// TIA Portal project "Ejercicio4-Proceso-TIA" (V14)

(* hardware
DEVICE "S7-1200 station_1"  S7-1200 Station
   slot 0: "Rack_0"  S7-1200 Rack  Rack  V1.0
   slot 1: "PLC_1"  CPU 1214C AC/DC/Rly  6ES7 214-1BG40-0XB0  V4.2
   slot 2: "AI 4x13BIT_1"  SM 1231 AI4  6ES7 231-4HD30-0XB0  V1.0
DEVICE "HMI_1"  TP 277 6''
   slot 0: "TP 277 6''"  TP 277 6''  6AV6 643-0AA01-1AX0  11.0.2.0
   slot 1: "HMI_RT_1"  TP 277 6''  6AV6 643-0AA01-1AX0  11.0.2.0
   slot 5: "HMI_1.IE_CP_1"  PROFINET Interface  11.0.0.0
      slot 1: "Interfaz PROFINET_1"  PROFINET Interface
         slot 1: "Port_1"  Port
   slot 7: "HMI_1.MPI/DP_CP_1"  MPI/DP Interface  11.0.0.0
*)

// ===== PLC "PLC_1"  CPU 1214C AC/DC/Rly =====

VAR_GLOBAL   // PLC tag table "Tabla de variables estándar"
   "System_Byte" AT %MB1 : Byte;
   "FirstScan" AT %M1.0 : Bool;
   "DiagStatusUpdate" AT %M1.1 : Bool;
   "AlwaysTRUE" AT %M1.2 : Bool;
   "AlwaysFALSE" AT %M1.3 : Bool;
   "System_Byte(1)" AT %MB1 : Byte;
   "Clock_Byte" AT %MB100 : Byte;
   "Clock_10Hz" AT %M100.0 : Bool;
   "Clock_5Hz" AT %M100.1 : Bool;
   "Clock_2.5Hz" AT %M100.2 : Bool;
   "Clock_2Hz" AT %M100.3 : Bool;
   "Clock_1.25Hz" AT %M100.4 : Bool;
   "Clock_1Hz" AT %M100.5 : Bool;
   "Clock_0.625Hz" AT %M100.6 : Bool;
   "Clock_0.5Hz" AT %M100.7 : Bool;
   "Tag_2" AT %MD8 : Real;
   "LT1" AT %IW30 : Int;
   "TT1" AT %IW100 : Int;
   "TT2" AT %IW102 : Int;
   "TT3" AT %IW104 : Int;
   "LT2" AT %IW98 : Int;
   "SLT1" AT %MD30 : Real;
   "SLT2" AT %MD38 : Real;
   "STT1" AT %MD46 : Real;
   "STT2" AT %MD54 : Real;
   "LedLT1" AT %Q0.0 : Bool;
   "LedLT2" AT %Q0.1 : Bool;
   "LedTT1" AT %Q0.2 : Bool;
   "LedTT2" AT %Q0.3 : Bool;
   "CorteDeLazo" AT %M0.5 : Bool;
   "START" AT %M0.0 : Bool;
   "STOP" AT %M0.1 : Bool;
   "Salida" AT %QD30 : Real;
   "Entrada" AT %ID2 : Real;
   "EncenderTanque" AT %ID6 : Real;
   "Ldl" AT %Q0.4 : Bool;
   "START/STOP" AT %M0.3 : Bool;
END_VAR

DATA_BLOCK "Transmisor TT1"   // DB1
{ S7_Optimized_Access := 'TRUE' }
VERSION : 0.1
// stored: InstanceOfName Escalado
"Escalado"
BEGIN
END_DATA_BLOCK

DATA_BLOCK "Transmisor TT2"   // DB2
{ S7_Optimized_Access := 'TRUE' }
VERSION : 0.1
// stored: InstanceOfName Escalado
"Escalado"
BEGIN
END_DATA_BLOCK

DATA_BLOCK "Transmisor LT1"   // DB3
{ S7_Optimized_Access := 'TRUE' }
VERSION : 0.1
// stored: InstanceOfName Escalado
"Escalado"
BEGIN
END_DATA_BLOCK

DATA_BLOCK "Transmisor LT2"   // DB4
{ S7_Optimized_Access := 'TRUE' }
VERSION : 0.1
// stored: InstanceOfName Escalado
"Escalado"
BEGIN
END_DATA_BLOCK

FUNCTION_BLOCK "Escalado"   // FB1, LAD
TITLE = Bloque de Escalado en Tension
{ S7_Optimized_Access := 'TRUE' }
VERSION : 0.1
   VAR_INPUT
      Entrada_IV : Int;
      ISH : Int;
      ISL : Int;
      OSH : Real;
      OSL : Real;
   END_VAR
   VAR_OUTPUT
      Salida : Real;
   END_VAR
   VAR_TEMP
      Temp_D : DInt;
      Temp_R : Real;
   END_VAR
BEGIN

REGION Network 1
   // (OSH - OSL)*(IV-ISL)/(ISH-ISL)+OSL
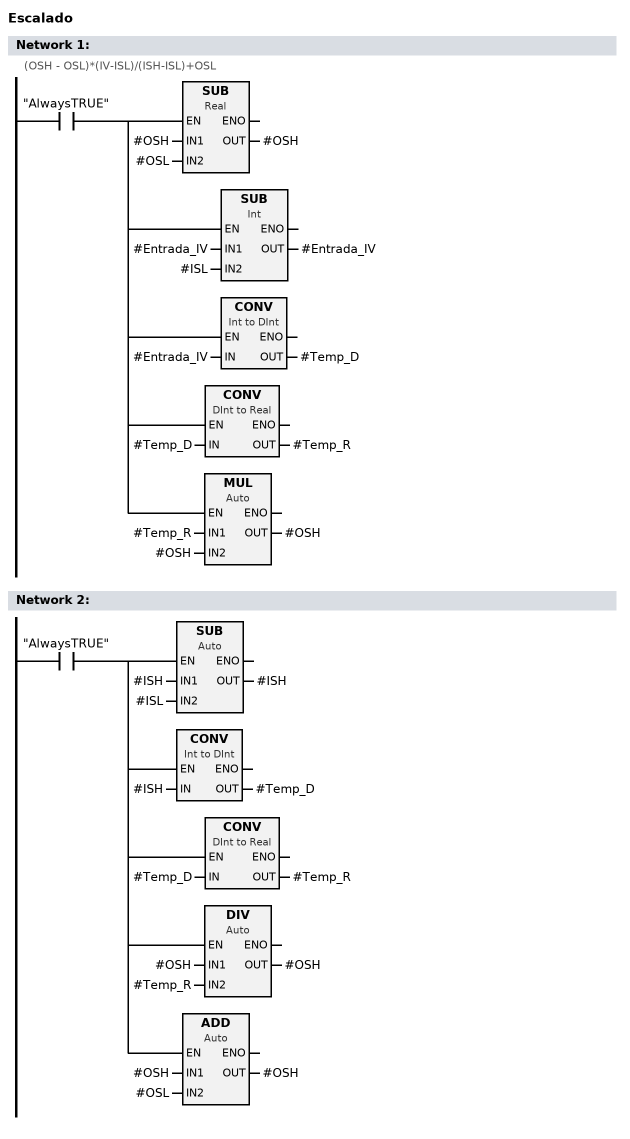
   RUNG wire#powerrail
      Contact( "AlwaysTRUE" )
      wire#w1
      { S7_Templates := "SrcType := Real" } Sub(in1 := #OSH, in2 := #OSL, out => #OSH)
   END_RUNG
   RUNG wire#w1
      { S7_Templates := "SrcType := Int" } Sub(in1 := #Entrada_IV, in2 := #ISL, out => #Entrada_IV)
   END_RUNG
   RUNG wire#w1
      { S7_Templates := "[SrcType := Int, DestType := DInt]" } Convert(in := #Entrada_IV, out => #Temp_D)
   END_RUNG
   RUNG wire#w1
      { S7_Templates := "[SrcType := DInt, DestType := Real]" } Convert(in := #Temp_D, out => #Temp_R)
   END_RUNG
   RUNG wire#w1
      Mul(in1 := #Temp_R, in2 := #OSH, out => #OSH)
   END_RUNG
   // the same network as SCL:
   IF "AlwaysTRUE" THEN
       #OSH := #OSH - #OSL;
       #Entrada_IV := #Entrada_IV - #ISL;
       #Temp_D := INT_TO_DINT(#Entrada_IV);
       #Temp_R := DINT_TO_REAL(#Temp_D);
       #OSH := #Temp_R * #OSH;
   END_IF;
END_REGION

REGION Network 2
   RUNG wire#powerrail
      Contact( "AlwaysTRUE" )
      wire#w1
      Sub(in1 := #ISH, in2 := #ISL, out => #ISH)
   END_RUNG
   RUNG wire#w1
      { S7_Templates := "[SrcType := Int, DestType := DInt]" } Convert(in := #ISH, out => #Temp_D)
   END_RUNG
   RUNG wire#w1
      { S7_Templates := "[SrcType := DInt, DestType := Real]" } Convert(in := #Temp_D, out => #Temp_R)
   END_RUNG
   RUNG wire#w1
      Div(in1 := #OSH, in2 := #Temp_R, out => #OSH)
   END_RUNG
   RUNG wire#w1
      Add(in1 := #OSH, in2 := #OSL, out => #OSH)
   END_RUNG
   // the same network as SCL:
   IF "AlwaysTRUE" THEN
       #ISH := #ISH - #ISL;
       #Temp_D := INT_TO_DINT(#ISH);
       #Temp_R := DINT_TO_REAL(#Temp_D);
       #OSH := #OSH / #Temp_R;
       #OSH := #OSH + #OSL;
   END_IF;
END_REGION
END_FUNCTION_BLOCK

FUNCTION "Alarmas" : Void   // FC1, LAD
TITLE = Alarmas
{ S7_Optimized_Access := 'TRUE' }
VERSION : 0.1
BEGIN

REGION Network 1: Alarmas por Corte de Lazo de corriente en transmisores de Nivel
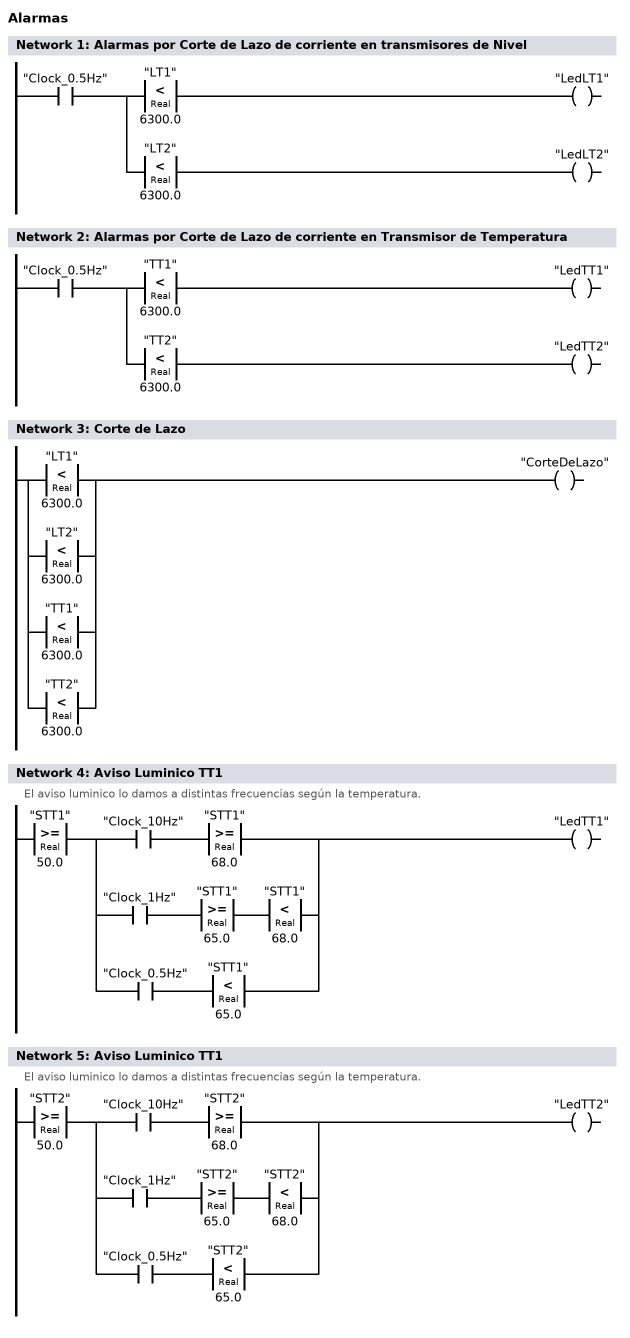
   RUNG wire#powerrail
      Contact( "Clock_0.5Hz" )
      wire#w1
      { S7_Templates := "SrcType := Real" } LT_Contact(in1 := "LT1", in2 := 6300.0)
      Coil( "LedLT1" )
   END_RUNG
   RUNG wire#w1
      { S7_Templates := "SrcType := Real" } LT_Contact(in1 := "LT2", in2 := 6300.0)
      Coil( "LedLT2" )
   END_RUNG
   // the same network as SCL:
   "LedLT1" := "Clock_0.5Hz" AND ("LT1" < 6300.0);
   "LedLT2" := "Clock_0.5Hz" AND ("LT2" < 6300.0);
END_REGION

REGION Network 2: Alarmas por Corte de Lazo de corriente en Transmisor de Temperatura
   RUNG wire#powerrail
      Contact( "Clock_0.5Hz" )
      wire#w1
      { S7_Templates := "SrcType := Real" } LT_Contact(in1 := "TT1", in2 := 6300.0)
      Coil( "LedTT1" )
   END_RUNG
   RUNG wire#w1
      { S7_Templates := "SrcType := Real" } LT_Contact(in1 := "TT2", in2 := 6300.0)
      Coil( "LedTT2" )
   END_RUNG
   // the same network as SCL:
   "LedTT1" := "Clock_0.5Hz" AND ("TT1" < 6300.0);
   "LedTT2" := "Clock_0.5Hz" AND ("TT2" < 6300.0);
END_REGION

REGION Network 3: Corte de Lazo
   RUNG wire#powerrail
      { S7_Templates := "SrcType := Real" } LT_Contact(in1 := "LT1", in2 := 6300.0)
      wire#w1
      Coil( "CorteDeLazo" )
   END_RUNG
   RUNG wire#powerrail
      { S7_Templates := "SrcType := Real" } LT_Contact(in1 := "LT2", in2 := 6300.0)
   END_RUNG wire#w1
   RUNG wire#powerrail
      { S7_Templates := "SrcType := Real" } LT_Contact(in1 := "TT1", in2 := 6300.0)
   END_RUNG wire#w1
   RUNG wire#powerrail
      { S7_Templates := "SrcType := Real" } LT_Contact(in1 := "TT2", in2 := 6300.0)
   END_RUNG wire#w1
   // the same network as SCL:
   "CorteDeLazo" := ("LT1" < 6300.0) OR ("LT2" < 6300.0) OR ("TT1" < 6300.0) OR ("TT2" < 6300.0);
END_REGION

REGION Network 4: Aviso Luminico TT1
   // El aviso luminico lo damos a distintas frecuencias según la temperatura.
   RUNG wire#powerrail
      { S7_Templates := "SrcType := Real" } GE_Contact(in1 := "STT1", in2 := 50.0)
      wire#w1
      Contact( "Clock_10Hz" )
      { S7_Templates := "SrcType := Real" } GE_Contact(in1 := "STT1", in2 := 68.0)
      wire#w2
      Coil( "LedTT1" )
   END_RUNG
   RUNG wire#w1
      Contact( "Clock_1Hz" )
      { S7_Templates := "SrcType := Real" } GE_Contact(in1 := "STT1", in2 := 65.0)
      { S7_Templates := "SrcType := Real" } LT_Contact(in1 := "STT1", in2 := 68.0)
   END_RUNG wire#w2
   RUNG wire#w1
      Contact( "Clock_0.5Hz" )
      { S7_Templates := "SrcType := Real" } LT_Contact(in1 := "STT1", in2 := 65.0)
   END_RUNG wire#w2
   // the same network as SCL:
   "LedTT1" := ("STT1" >= 50.0) AND (("Clock_10Hz" AND ("STT1" >= 68.0)) OR ("Clock_1Hz" AND ("STT1" >= 65.0) AND ("STT1" < 68.0)) OR ("Clock_0.5Hz" AND ("STT1" < 65.0)));
END_REGION

REGION Network 5: Aviso Luminico TT1
   // El aviso luminico lo damos a distintas frecuencias según la temperatura.
   RUNG wire#powerrail
      { S7_Templates := "SrcType := Real" } GE_Contact(in1 := "STT2", in2 := 50.0)
      wire#w1
      Contact( "Clock_10Hz" )
      { S7_Templates := "SrcType := Real" } GE_Contact(in1 := "STT2", in2 := 68.0)
      wire#w2
      Coil( "LedTT2" )
   END_RUNG
   RUNG wire#w1
      Contact( "Clock_1Hz" )
      { S7_Templates := "SrcType := Real" } GE_Contact(in1 := "STT2", in2 := 65.0)
      { S7_Templates := "SrcType := Real" } LT_Contact(in1 := "STT2", in2 := 68.0)
   END_RUNG wire#w2
   RUNG wire#w1
      Contact( "Clock_0.5Hz" )
      { S7_Templates := "SrcType := Real" } LT_Contact(in1 := "STT2", in2 := 65.0)
   END_RUNG wire#w2
   // the same network as SCL:
   "LedTT2" := ("STT2" >= 50.0) AND (("Clock_10Hz" AND ("STT2" >= 68.0)) OR ("Clock_1Hz" AND ("STT2" >= 65.0) AND ("STT2" < 68.0)) OR ("Clock_0.5Hz" AND ("STT2" < 65.0)));
END_REGION
END_FUNCTION

FUNCTION "Control_Temperatura" : Void   // FC2, LAD
{ S7_Optimized_Access := 'TRUE' }
VERSION : 0.1
BEGIN

REGION Network 1
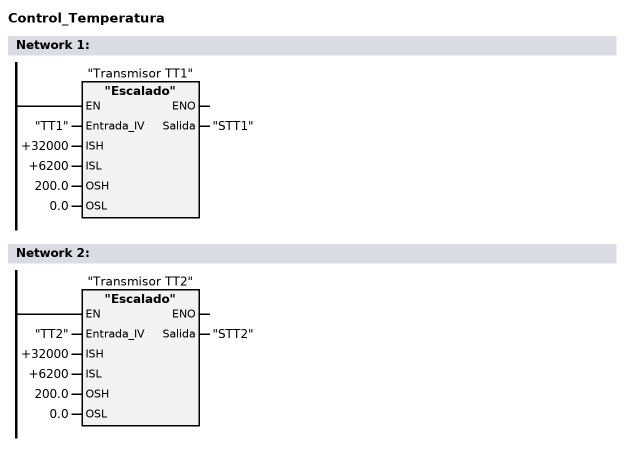
   RUNG wire#powerrail
      "Transmisor TT1"(Entrada_IV := "TT1", ISH := +32000, ISL := +6200, OSH := 200.0, OSL := 0.0, Salida => "STT1")
   END_RUNG
   // the same network as SCL:
   "Transmisor TT1"(Entrada_IV := "TT1",   // "Escalado"
                    ISH := +32000,
                    ISL := +6200,
                    OSH := 200.0,
                    OSL := 0.0,
                    Salida => "STT1");
END_REGION

REGION Network 2
   RUNG wire#powerrail
      "Transmisor TT2"(Entrada_IV := "TT2", ISH := +32000, ISL := +6200, OSH := 200.0, OSL := 0.0, Salida => "STT2")
   END_RUNG
   // the same network as SCL:
   "Transmisor TT2"(Entrada_IV := "TT2",   // "Escalado"
                    ISH := +32000,
                    ISL := +6200,
                    OSH := 200.0,
                    OSL := 0.0,
                    Salida => "STT2");
END_REGION
END_FUNCTION

FUNCTION "Control_Nivel" : Void   // FC3, LAD
{ S7_Optimized_Access := 'TRUE' }
VERSION : 0.1
BEGIN

REGION Network 1
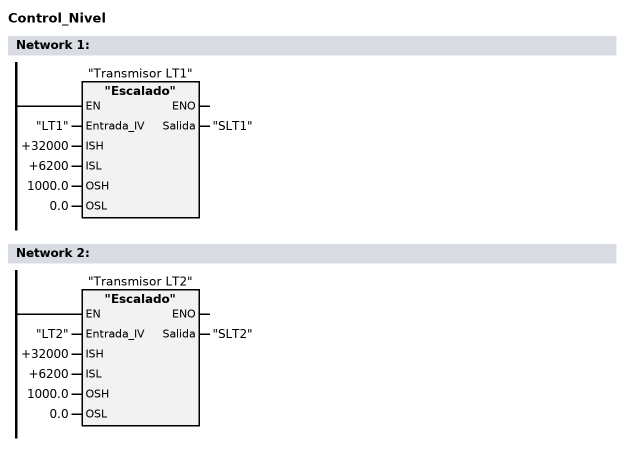
   RUNG wire#powerrail
      "Transmisor LT1"(Entrada_IV := "LT1", ISH := +32000, ISL := +6200, OSH := 1000.0, OSL := 0.0, Salida => "SLT1")
   END_RUNG
   // the same network as SCL:
   "Transmisor LT1"(Entrada_IV := "LT1",   // "Escalado"
                    ISH := +32000,
                    ISL := +6200,
                    OSH := 1000.0,
                    OSL := 0.0,
                    Salida => "SLT1");
END_REGION

REGION Network 2
   RUNG wire#powerrail
      "Transmisor LT2"(Entrada_IV := "LT2", ISH := +32000, ISL := +6200, OSH := 1000.0, OSL := 0.0, Salida => "SLT2")
   END_RUNG
   // the same network as SCL:
   "Transmisor LT2"(Entrada_IV := "LT2",   // "Escalado"
                    ISH := +32000,
                    ISL := +6200,
                    OSH := 1000.0,
                    OSL := 0.0,
                    Salida => "SLT2");
END_REGION
END_FUNCTION

FUNCTION "EncenderParar" : Void   // FC4, LAD
{ S7_Optimized_Access := 'TRUE' }
VERSION : 0.1
BEGIN

REGION Network 1
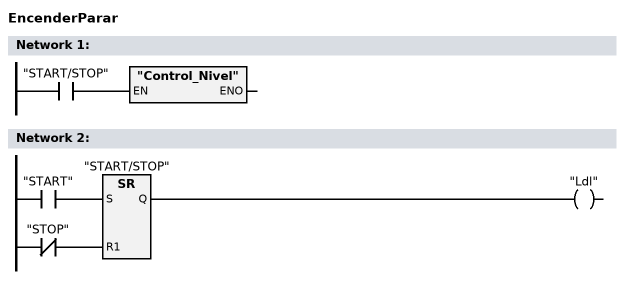
   RUNG wire#powerrail
      Contact( "START/STOP" )
      "Control_Nivel"()
   END_RUNG
   // the same network as SCL:
   IF "START/STOP" THEN "Control_Nivel"(); END_IF;
END_REGION

REGION Network 2
   RUNG wire#powerrail
      Contact( "START" )
      S_SR(operand := "START/STOP", r1 := wire#w1)
      Coil( "Ldl" )
   END_RUNG
   RUNG wire#powerrail
      I_Contact( "STOP" )
   END_RUNG wire#w1
   // the same network as SCL:
   IF "START" THEN
       "START/STOP" := TRUE;   // SR flip-flop
   END_IF;
   IF NOT "STOP" THEN "START/STOP" := FALSE; END_IF;
   "Ldl" := "START/STOP";
END_REGION
END_FUNCTION

ORGANIZATION_BLOCK "Main"   // OB1, LAD, ProgramCycle
TITLE = "Main Program Sweep (Cycle)"
{ S7_Optimized_Access := 'TRUE' }
VERSION : 0.1
   VAR_INPUT
      Initial_Call : Bool;   // Initial call of this OB
      Remanence : Bool;   // =True, if remanent data are available
   END_VAR
BEGIN

REGION Network 1
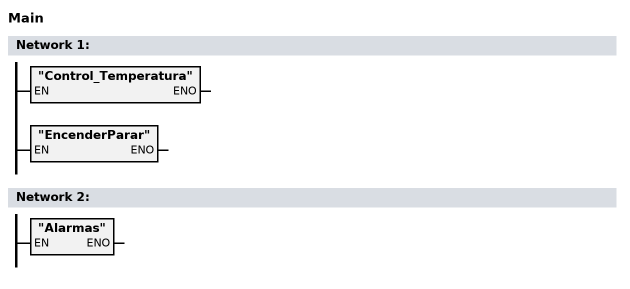
   RUNG wire#powerrail
      "Control_Temperatura"()
   END_RUNG
   RUNG wire#powerrail
      "EncenderParar"()
   END_RUNG
   // the same network as SCL:
   "Control_Temperatura"();
   "EncenderParar"();
END_REGION

REGION Network 2
   RUNG wire#powerrail
      "Alarmas"()
   END_RUNG
   // the same network as SCL:
   "Alarmas"();
END_REGION
END_ORGANIZATION_BLOCK

(* ===== HMI "HMI_RT_1" =====
system functions are stored by id; their names below are inferred from use
connection "HMI_Conexión_1": ETHERNET, SIMATIC S7 1200

HMI tags "Tabla de variables estándar"
   "START" : Bool = PLC START AT %M0.0, 1 s
   "STOP" : Bool = PLC STOP AT %M0.1, 1 s
   "START-STOP" : Bool = PLC "START/STOP" AT %M0.3, 1 s
   "LedLT1" : Bool = PLC LedLT1 AT %Q0.0, 1 s
   "LedLT2" : Bool = PLC LedLT2 AT %Q0.1, 1 s
   "LedTT1" : Bool = PLC LedTT1 AT %Q0.2, 1 s
   "LedTT2" : Bool = PLC LedTT2 AT %Q0.3, 1 s
   "LT1" : Int = PLC LT1 AT %IW30, 1 s
   "LT2" : Int = PLC LT2 AT %IW98, 1 s
   "TT1" : Int = PLC TT1 AT %IW100, 1 s
   "TT2" : Int = PLC TT2 AT %IW102, 1 s
   "SLT1" : Real = PLC SLT1 AT %MD30, 1 s
   "SLT2" : Real = PLC SLT2 AT %MD38, 1 s
   "STT1" : Real = PLC STT1 AT %MD46, 1 s
   "STT2" : Real = PLC STT2 AT %MD54, 1 s
   "CortedeLazo" : Bool = PLC CorteDeLazo AT %M0.5, 1 s

screen "MENU-INDICADORESLEDS" 320x240
   Button "Botón_1" at 213,47 size 96x30; TextOff 'Encender'
      on Click: SetBit("START"); SetBit("STOP")
   Button "Botón_2" at 213,83 size 96x30; TextOff 'Apagar'
      on Click: ResetBit("START"); ResetBit("STOP")
   Rectangle "Rectángulo_1" at 16,31 size 48x24
      Appearance <- "START-STOP"
   Rectangle "Rectángulo_2" at 16,71 size 48x24
      Appearance <- "LedLT1"
   Rectangle "Rectángulo_3" at 16,111 size 48x24
      Appearance <- "LedLT2"
   Rectangle "Rectángulo_4" at 16,151 size 48x24
      Appearance <- "LedTT1"
   Rectangle "Rectángulo_5" at 16,188 size 48x24
      Appearance <- "LedTT2"
   Rectangle "Rectángulo_6" at 281,212 size 26x24
      Appearance <- "CortedeLazo"
   TextField "Campo de texto_1" at 177,213 size 95x18; Text 'Corte de Lazo'
   TextField "Campo de texto_2" at 16,13 size 46x18; Text 'ON/Off'
   TextField "Campo de texto_3" at 16,53 size 25x18; Text 'LT1'
   TextField "Campo de texto_4" at 17,93 size 25x18; Text 'LT2'
   TextField "Campo de texto_5" at 17,133 size 25x18; Text 'TT1'
   TextField "Campo de texto_6" at 17,173 size 25x18; Text 'TT1'
   Button "Botón_3" at 212,121 size 96x30; TextOff 'Nivel'
      on Click: ActivateScreen("NIVEL", 0)
   Button "Botón_4" at 212,156 size 96x30; TextOff 'Temperatura'
      on Click: ActivateScreen("TEMPERATURA", 0)

screen "NIVEL" 320x240
   Bar "Barra_1" at 3,7 size 158x178; MinimumValue 0; MaximumValue 100
      ProcessValue <- "SLT1"
   Bar "Barra_2" at 161,7 size 158x178; MinimumValue 0; MaximumValue 100
      ProcessValue <- "SLT2"
   Button "Botón_1" at 218,205 size 95x31; TextOff 'Temperatura'
      on Click: ActivateScreen("TEMPERATURA", 0)
   Button "Botón_2" at 7,205 size 95x31; TextOff 'Menu'
      on Click: ActivateScreen("MENU-INDICADORESLEDS", 0)
   TextField "Campo de texto_1" at 50,180 size 29x20; Text 'LT1'
   TextField "Campo de texto_2" at 213,180 size 29x20; Text 'LT2'

screen "TEMPERATURA" 320x240
   Gauge "Indicador gauge_1" at 0,0 size 158x158; CaptionText 'SIMATIC'
      ProcessValue <- "SLT1"
   Gauge "Indicador gauge_2" at 160,0 size 158x158; CaptionText 'SIMATIC'
      ProcessValue <- "LedTT2"
   Button "Botón_3" at 218,205 size 95x31; TextOff 'Nivel'
      on Click: ActivateScreen("NIVEL", 0)
   Button "Botón_1" at 7,205 size 95x31; TextOff 'Menu'
      on Click: ActivateScreen("MENU-INDICADORESLEDS", 0)
   TextField "Campo de texto_1" at 65,158 size 29x20; Text 'TT1'
   TextField "Campo de texto_2" at 227,158 size 29x20; Text 'TT2'
*)